ABB RobotStudio station: Solution2_Gripper_Hicham.rspag

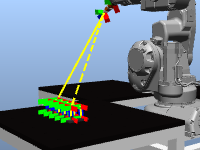
--- station ---
Station Solution3 (saved by RobotStudio 7.0.8504.151)
Controller IRB_140_6kg_0.81m, task T_ROB1: task frame (RAPID world) sits at (0, 0, 670) mm in the station
Controller IRB_140_6kg_0.81m
  mechanical unit ROB_1: IRB140_6_81_C_03, 6 joints, base frame (0, 0, 0) mm
Layout (positions relative to the parent item):
  - IRB140_6_81_C_03 [mechanism, from Robots\IRB140_6_81_C_G_03.rslib] at (0, 0, 670) mm; joint values [0, 0, 0, 0, 0.5236, 0] (rad or m)
  - gripper2 [mechanism, from RobotStudio_RW603_files_Lab2_Gripper\gripper.rslib] at (506.29, 0, 1349.5) mm, rotated rx 180 ry 60 rz 180 deg; joint values [0] (rad or m)
  - piece12 [part, from RobotStudio_RW603_files_Lab2_Gripper\piece12.rslib] at (100, 675, 798) mm
  - piece12_2 [part, from RobotStudio_RW603_files_Lab2_Gripper\piece12.rslib] at (150, 675, 798) mm
  - piece12_3 [part, from RobotStudio_RW603_files_Lab2_Gripper\piece12.rslib] at (50, 671.5, 798) mm
  - piece12_4 [part, from RobotStudio_RW603_files_Lab2_Gripper\piece12.rslib] at (0, 671.5, 798) mm
  - piece12_5 [part, from RobotStudio_RW603_files_Lab2_Gripper\piece12.rslib] at (-50, 671.5, 798) mm
  - rob-table [part, from RobotStudio_RW603_files_Lab2_Gripper\rob-table.rslib]
  - brick [part, from RobotStudio_RW603_files_Lab2_Gripper\brick.rslib] at (175, 600, 790) mm
Attachment: gripper2 is attached to IRB140_6_81_C_03 / Link6
EventTableEntry 1099: Group=, Trigger=DO10_1 1100, Actions=[EventTableActionAttach 1101], Comment=, ActivationMode=2, Cyclic=false
EventTableTriggerIO 1100: IOValue=[1], IRC5Controller=? -1, Operator=0, SignalSource=IRB_140_6kg_0.81m 491
EventTableActionAttach 1101: AttachmentParent=gripper2 983, AttachmentChild=? -1, MountObject=false, Offset=[X=1, Y=0, Z=0, W=0, X=0, Y=1, Z=0, W=0, X=0, Y=0, Z=1, W=0, X=0, Y=0, Z=0, W=1], FlangeIndext=0, FindNearest=true
EventTableEntry 1102: Group=, Trigger=DO10_0 1103, Actions=[EventTableActionDetach 1104], Comment=, ActivationMode=2, Cyclic=false
EventTableTriggerIO 1103: IOValue=[1], IRC5Controller=? -1, Operator=0, SignalSource=IRB_140_6kg_0.81m 491
EventTableActionDetach 1104: AttachmentParent=gripper2 983, AttachmentChild=? -1

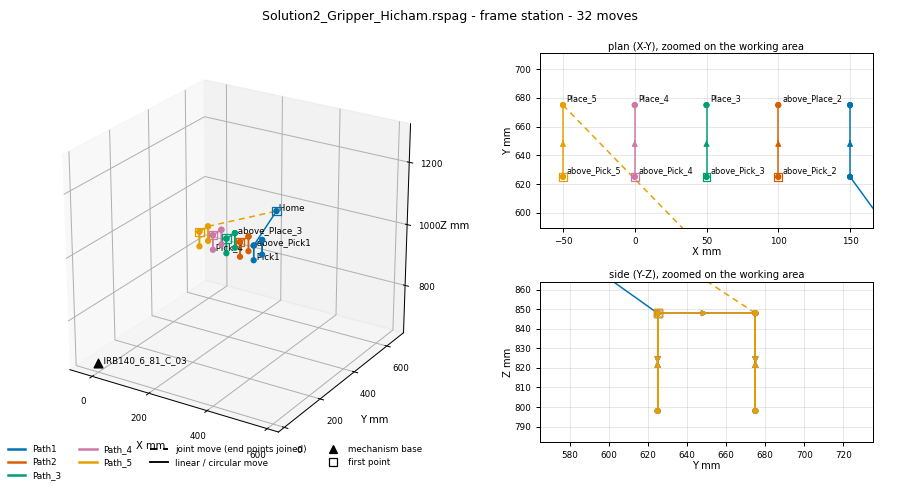
[picture p0: tool path of Solution2_Gripper_Hicham.rspag in frame station, 32 of 32 moves have a stored position in this frame; points joined in program order, loops and branches not executed]
--- Backups/IRB_140_6kg_0.81m/RAPID/TASK1/PROGMOD/CalibData.mod ---
MODULE CalibData
	PERS tooldata gripper:=[TRUE,[[0,0,115],[1,0,0,0]],[0.5,[0,0,30],[1,0,0,0],0,0,0]];
	TASK PERS wobjdata Workobject_1:=[FALSE,TRUE,"",[[175,600,120],[0,0,1,0]],[[25,25,-8],[1,0,0,0]]];
ENDMODULE

--- Backups/IRB_140_6kg_0.81m/RAPID/TASK1/PROGMOD/Module1.mod ---
MODULE Module1
	CONST robtarget Home:=[[-455.884572681,-625,-494],[0.866025404,0,-0.5,0],[0,0,0,0],[9E+09,9E+09,9E+09,9E+09,9E+09,9E+09]];

    CONST robtarget Pick1:=[[0,0,0],[1,0,0,0],[0,0,0,0],[9E+09,9E+09,9E+09,9E+09,9E+09,9E+09]];
    CONST robtarget above_Pick1:=[[0,0,-50],[1,0,0,0],[0,0,0,0],[9E+09,9E+09,9E+09,9E+09,9E+09,9E+09]];
    CONST robtarget above_Place1_10:=[[0,50,-50],[1,0,0,0],[0,0,0,0],[9E+09,9E+09,9E+09,9E+09,9E+09,9E+09]];
    CONST robtarget Place1:=[[0,50,0],[1,0,0,0],[0,0,0,0],[9E+09,9E+09,9E+09,9E+09,9E+09,9E+09]];
    CONST robtarget above_Place1:=[[0,50,-50],[1,0,0,0],[0,0,0,0],[9E+09,9E+09,9E+09,9E+09,9E+09,9E+09]];

    CONST robtarget above_Pick_2:=[[50,0,-50],[1,0,0,0],[0,0,0,0],[9E+09,9E+09,9E+09,9E+09,9E+09,9E+09]];
    CONST robtarget Pick_2:=[[50,0,0],[1,0,0,0],[0,0,0,0],[9E+09,9E+09,9E+09,9E+09,9E+09,9E+09]];
    CONST robtarget above_Place_2:=[[50,50,-50],[1,0,0,0],[0,0,0,0],[9E+09,9E+09,9E+09,9E+09,9E+09,9E+09]];
    CONST robtarget Place_2:=[[50,50,0],[1,0,0,0],[0,0,0,0],[9E+09,9E+09,9E+09,9E+09,9E+09,9E+09]];

    CONST robtarget above_Pick_3:=[[100,0,-50],[1,0,0,0],[1,0,0,0],[9E+09,9E+09,9E+09,9E+09,9E+09,9E+09]];
    CONST robtarget Pick_3:=[[100,0,0],[1,0,0,0],[1,0,0,0],[9E+09,9E+09,9E+09,9E+09,9E+09,9E+09]];
    CONST robtarget above_Place_3:=[[100,50,-50],[1,0,0,0],[1,0,0,0],[9E+09,9E+09,9E+09,9E+09,9E+09,9E+09]];
    CONST robtarget Place_3:=[[100,50,0],[1,0,0,0],[1,0,0,0],[9E+09,9E+09,9E+09,9E+09,9E+09,9E+09]];

    CONST robtarget above_Pick_4:=[[150,0,-50],[1,0,0,0],[1,0,0,0],[9E+09,9E+09,9E+09,9E+09,9E+09,9E+09]];
    CONST robtarget Pick_4:=[[150,0,0],[1,0,0,0],[1,0,0,0],[9E+09,9E+09,9E+09,9E+09,9E+09,9E+09]];
    CONST robtarget above_Place_4:=[[150,50,-50],[1,0,0,0],[1,0,0,0],[9E+09,9E+09,9E+09,9E+09,9E+09,9E+09]];
    CONST robtarget Place_4:=[[150,50,0],[1,0,0,0],[1,0,0,0],[9E+09,9E+09,9E+09,9E+09,9E+09,9E+09]];

    CONST robtarget above_Pick_5:=[[200,0,-50],[1,0,0,0],[1,0,1,0],[9E+09,9E+09,9E+09,9E+09,9E+09,9E+09]];
    CONST robtarget Pick_5:=[[200,0,0],[1,0,0,0],[1,0,1,0],[9E+09,9E+09,9E+09,9E+09,9E+09,9E+09]];
    CONST robtarget above_Place_5:=[[200,50,-50],[1,0,0,0],[1,0,1,0],[9E+09,9E+09,9E+09,9E+09,9E+09,9E+09]];
    CONST robtarget Place_5:=[[200,50,0],[1,0,0,0],[1,0,1,0],[9E+09,9E+09,9E+09,9E+09,9E+09,9E+09]];


	PROC main()
	    Path1;
        Path2;
        Path_3;
        Path_4;
        Path_5;
	ENDPROC
    PROC Path1()
        MoveJ Home,v100,z100,gripper\WObj:=Workobject_1;
        SetDO DO10_0,1;
        SetDO DO10_1,0;
        WaitTime 2;
        MoveL above_Pick1,v100,z10,gripper\WObj:=Workobject_1;
        MoveL Pick1,v100,fine,gripper\WObj:=Workobject_1;
        WaitTime 2;
        ! set the digital outputs to CLOSE the gripper
        SetDO DO10_0,0;
        SetDO DO10_1,1;
        WaitTime 2;
        MoveL above_Pick1,v100,z10,gripper\WObj:=Workobject_1;
        MoveL above_Place1,v100,z10,gripper\WObj:=Workobject_1;
        MoveL Place1,v100,fine,gripper\WObj:=Workobject_1;
        WaitTime 2;
        ! set the digital outputs to OPEN the gripper
        SetDO DO10_0,1;
        SetDO DO10_1,0;
        WaitTime 2;
        MoveL above_Place1,v100,z10,gripper\WObj:=Workobject_1;
    ENDPROC
    PROC Path2()
        MoveL above_Pick_2,v100,z10,gripper\WObj:=Workobject_1;
        MoveL Pick_2,v100,fine,gripper\WObj:=Workobject_1;
        WaitTime 2;
        ! set the digital outputs to CLOSE the gripper
        SetDO DO10_0,0;
        SetDO DO10_1,1;
        WaitTime 2;
        MoveL above_Pick_2,v100,z10,gripper\WObj:=Workobject_1;
        MoveL above_Place_2,v100,z10,gripper\WObj:=Workobject_1;
        MoveL Place_2,v100,fine,gripper\WObj:=Workobject_1;
        WaitTime 2;
        ! set the digital outputs to OPEN the gripper
        SetDO DO10_0,1;
        SetDO DO10_1,0;
        WaitTime 2;
        MoveL above_Place_2,v100,z10,gripper\WObj:=Workobject_1;
    ENDPROC
    PROC Path_3()
        MoveL above_Pick_3,v100,z10,gripper\WObj:=Workobject_1;
        MoveL Pick_3,v100,fine,gripper\WObj:=Workobject_1;
        WaitTime 2;
        ! set the digital outputs to CLOSE the gripper
        SetDO DO10_0,0;
        SetDO DO10_1,1;
        WaitTime 2;
        MoveL above_Pick_3,v100,z10,gripper\WObj:=Workobject_1;
        MoveL above_Place_3,v100,z10,gripper\WObj:=Workobject_1;
        MoveL Place_3,v100,fine,gripper\WObj:=Workobject_1;
        WaitTime 2;
        ! set the digital outputs to OPEN the gripper
        SetDO DO10_0,1;
        SetDO DO10_1,0;
        WaitTime 2;
        MoveL above_Place_3,v100,z10,gripper\WObj:=Workobject_1;
    ENDPROC
    PROC Path_4()
        MoveL above_Pick_4,v100,z10,gripper\WObj:=Workobject_1;
        MoveL Pick_4,v100,fine,gripper\WObj:=Workobject_1;
        WaitTime 2;
        ! set the digital outputs to CLOSE the gripper
        SetDO DO10_0,0;
        SetDO DO10_1,1;
        WaitTime 2;
        MoveL above_Pick_4,v100,z10,gripper\WObj:=Workobject_1;
        MoveL above_Place_4,v100,z10,gripper\WObj:=Workobject_1;
        MoveL Place_4,v100,fine,gripper\WObj:=Workobject_1;
        WaitTime 2;
        ! set the digital outputs to OPEN the gripper
        SetDO DO10_0,1;
        SetDO DO10_1,0;
        WaitTime 2;
        MoveL above_Place_4,v100,z10,gripper\WObj:=Workobject_1;
    ENDPROC
    PROC Path_5()
        MoveL above_Pick_5,v100,z10,gripper\WObj:=Workobject_1;
        MoveL Pick_5,v100,fine,gripper\WObj:=Workobject_1;
        WaitTime 2;
        ! set the digital outputs to CLOSE the gripper
        SetDO DO10_0,0;
        SetDO DO10_1,1;
        WaitTime 2;
        MoveL above_Pick_5,v100,z10,gripper\WObj:=Workobject_1;
        MoveL above_Place_5,v100,z10,gripper\WObj:=Workobject_1;
        MoveL Place_5,v100,fine,gripper\WObj:=Workobject_1;
        WaitTime 2;
        ! set the digital outputs to OPEN the gripper
        SetDO DO10_0,1;
        SetDO DO10_1,0;
        WaitTime 2;
        MoveL above_Place_5,v100,z10,gripper\WObj:=Workobject_1;
        MoveJ Home,v1000,z100,gripper\WObj:=Workobject_1;
    ENDPROC

ENDMODULE

--- Backups/IRB_140_6kg_0.81m/SYSPAR/EIO.cfg ---
EIO:CFG_1.0:6:1::
#
EIO_SIGNAL:

      -Name "DO10_0" -SignalType "DO"

      -Name "DO10_1" -SignalType "DO" -Default 1
